{attribute addProperty BoxType "EL2535-0103-0023"}
{attribute addProperty Id "StatusAT %I*Status_D7D8B361162"}
{attribute addProperty CRC "502109842"}
{attribute addProperty SizeInBites "16"}
{attribute addProperty SizeInBytes "2"}
TYPE PWM_Status_Channel_1DED9692 :
STRUCT
	{attribute addProperty Name "Status"}
	Status AT %I* : Status_D7D8B361;
END_STRUCT
END_TYPE

(* stored: Version 1.2.0.0, ProductVersion 3.1.4024.9
   DUT PWM_Status_Channel_1DED9692: Id {98675c97-86d0-40ec-9ac9-855070e8fe80} *)
